(*********************************** G.D S.p.A. - Technical Department ***********************************
============= PROGRAM INFO ============
FOLDER:             TBD
MACHINES INVOLVED:  TBD 

============= DESCRIPTION =============
csp machine declaration

============= REVISIONS ===============
Date		Version	 	Author      	Description             
----------	-------		------------  	--------------------------------------------
2019/04/05 	0000.00	 	M.Grasso		Creation of the PRG

**********************************************************************************************************)
(*$R process_ref := prc; $*)
PROGRAM csp_case_feed_reject
VAR
		
	prc:											process;
	prc_path:										STRING;
	
END_VAR

_read_var_input();

_object_manager();

IF NOT objects_running()
THEN
	RETURN;	
END_IF

_read_process_image();

_mode_manager();

_set_runtime_properties();

(********************************* BODY *********************************)
(************************************************************************)

_handle_messages();

_write_output();

ACTION _handle_messages:
;
END_ACTION

ACTION _handle_process_test:
;
END_ACTION

ACTION _mode_manager:
IF process_mode_req_is_pending(prc)
THEN
    process_apply_mode_req_first_step(prc);
    CASE process_get_mode(prc) OF
        MODE_TO_ABSENT:
			;
        MODE_TO_INACTIVE:
			;
        MODE_TO_TEST:
			;
        MODE_TO_OPERATIONAL:
			;
    END_CASE
    process_apply_mode_req_second_step(prc);
END_IF
END_ACTION

ACTION _object_manager:
IF objects_initialization()
THEN
	sub_process_init(
		object_name					:= 'csp_case_feed_reject.prc', 
		process						:= csp_case_feed.prc, 
		CONVERSION_this				:= prc);
		
	prc_path 						:= process_get_path(prc);
END_IF

IF objects_running()
THEN
	process_cycle(prc);
END_IF
END_ACTION

ACTION _read_process_image:
;
END_ACTION

ACTION _read_var_input:
;
END_ACTION

ACTION _set_runtime_properties:
;
END_ACTION

ACTION _write_output:
;
END_ACTION

END_PROGRAM

(* stored: Version 1.1.0.1, ProductVersion 3.1.4022.12
   POU csp_case_feed_reject: Id {c31a09c0-d733-430d-98e3-1616a1961183}, SpecialFunc None
   Action _handle_messages: Id {04ac5c31-203a-4c21-ad50-7a295370dbc2}
   Action _handle_process_test: Id {1c93239a-2e88-4433-a079-8a6a4c3fca00}
   Action _mode_manager: Id {0f95a701-ccdf-45f2-bd51-4df35e5f0b0e}
   Action _object_manager: Id {21f82159-b8d6-46f2-aaa6-dfba7f10c25d}
   Action _read_process_image: Id {3d340df3-e7c0-4879-a04a-6118e96f8f82}
   Action _read_var_input: Id {fde26385-4efd-43ea-a3a2-197e527bea7c}
   Action _set_runtime_properties: Id {fdc12529-3fd1-42f9-a76f-2c6c68b092bc}
   Action _write_output: Id {56faa11e-127e-4481-9143-85a7010cc191} *)
